FUNCTION_BLOCK fbValueSimulation
VAR_INPUT
	MinValue : REAL;
	MaxValue : REAL;
END_VAR
VAR_OUTPUT
	Value : REAL;
END_VAR
VAR
	rn : DRAND;
END_VAR

rn();

Value := LREAL_TO_REAL(MinValue + rn.Num * (MaxValue-MinValue));

END_FUNCTION_BLOCK

(* stored: Version 1.1.0.1, ProductVersion 3.1.4024.2
   POU fbValueSimulation: Id {c7732cf4-431d-4422-8f53-ab53ba420281}, SpecialFunc None *)
